INTERFACE IACVariobatch EXTENDS IACComponent

PROPERTY InSimulation : BOOL
GET
END_GET
END_PROPERTY

METHOD OnObjectMetaBuilded
VAR_INPUT
	iObject : IACObject;
END_VAR
END_METHOD

METHOD OnPropertyChangedBool
VAR_INPUT
	object : IACObject;
	propertyID : UINT;
	value : BOOL;
END_VAR
END_METHOD

METHOD OnPropertyChangedByte
VAR_INPUT
	object : IACObject;
	propertyID : UINT;
	value : BYTE;
END_VAR
END_METHOD

METHOD OnPropertyChangedDInt
VAR_INPUT
	object : IACObject;
	propertyID : UINT;
	value : DINT;
END_VAR
END_METHOD

METHOD OnPropertyChangedDT
VAR_INPUT
	object : IACObject;
	propertyID : UINT;
	value : DATE_AND_TIME;
END_VAR
END_METHOD

METHOD OnPropertyChangedInt
VAR_INPUT
	object : IACObject;
	propertyID : UINT;
	value : INT;
END_VAR
END_METHOD

METHOD OnPropertyChangedLReal
VAR_INPUT
	object : IACObject;
	propertyID : UINT;
	value : LREAL;
END_VAR
END_METHOD

METHOD OnPropertyChangedReal
VAR_INPUT
	object : IACObject;
	propertyID : UINT;
	value : REAL;
END_VAR
END_METHOD

METHOD OnPropertyChangedString
VAR_INPUT
	object : IACObject;
	propertyID : UINT;
	value : STRING(255);
END_VAR
END_METHOD

METHOD OnPropertyChangedTime
VAR_INPUT
	object : IACObject;
	propertyID : UINT;
	value : TIME;
END_VAR
END_METHOD

METHOD OnPropertyChangedUDInt
VAR_INPUT
	object : IACObject;
	propertyID : UINT;
	value : UDINT;
END_VAR
END_METHOD

METHOD OnPropertyChangedUInt
VAR_INPUT
	object : IACObject;
	propertyID : UINT;
	value : UINT;
END_VAR
END_METHOD

METHOD SetCompMetadata
VAR_INPUT
	iObject : IACObject;
END_VAR
END_METHOD

METHOD SetPropMetadata
VAR_INPUT
	iObject : IACObject;
	propertyID : UINT;
	sizeOfPropType : UINT;
END_VAR
END_METHOD

END_INTERFACE

(* stored: Version 1.1.0.1, ProductVersion 3.1.4022.7
   Itf IACVariobatch: Id {8eb91f6a-0d40-40db-9547-9c649a6bda0c}
   Property InSimulation: Id {367b4412-c9f5-4080-9eb4-5617b17b1b25}
   Get Get: Id {647f0321-8baf-45e1-a51d-10442fba99c6}
   Method OnObjectMetaBuilded: Id {b55e04eb-7cf5-4bf7-89ad-d490ce8a828e}
   Method OnPropertyChangedBool: Id {1776999f-6a53-4697-8545-f7bd4166d2db}
   Method OnPropertyChangedByte: Id {d577379f-2829-410b-92c8-c1d8b4fb2882}
   Method OnPropertyChangedDInt: Id {71c3db3a-ccf6-44f6-a368-ce0b17e2d3b1}
   Method OnPropertyChangedDT: Id {dce067c7-cb47-4d1f-bcb7-56f3ae3abdff}
   Method OnPropertyChangedInt: Id {dfb2a76b-81d5-46d6-b9f4-3a0c5cf1bfd3}
   Method OnPropertyChangedLReal: Id {a9d5e860-7e92-4555-9854-5852c8cde573}
   Method OnPropertyChangedReal: Id {685de739-9991-468a-9138-7e6faea786d5}
   Method OnPropertyChangedString: Id {7e0fb65b-6359-459a-adbc-fbe0ed4cd4c8}
   Method OnPropertyChangedTime: Id {8c610fe7-32e1-4aae-81fb-7a76b9315f99}
   Method OnPropertyChangedUDInt: Id {398cd77a-45cc-4191-92fe-b0fb4f111d77}
   Method OnPropertyChangedUInt: Id {45067c66-fa21-49cf-a647-7e6355472669}
   Method SetCompMetadata: Id {b0414800-dd55-4d67-98b5-90fa0672366d}
   Method SetPropMetadata: Id {34245123-aeab-489c-949b-701c041042c1} *)
